{attribute 'GeneratedUsingTerminal: EL3314-0002-0016'}
{attribute addProperty BoxType "EL3314-0002-0016"}
{attribute addProperty Id "TC_Inputs_Channel_1AT %I*TC_Inputs_Channel_4521310411TC_Inputs_Channel_2AT %I*TC_Inputs_Channel_4521310411TC_Inputs_Channel_3AT %I*TC_Inputs_Channel_4521310411TC_Inputs_Channel_4AT %I*TC_Inputs_Channel_4521310411WcStateAT %I*WcState_9091E0EB2InfoDataAT %I*InfoData_94A18F5E2"}
{attribute addProperty CRC "1814089623"}
{attribute addProperty Size "48"}
TYPE EL3314_6C20CF97 EXTENDS EtcSlaveTerminalBase_947E5A46 :
STRUCT
	{attribute addProperty Name "TC_Inputs_Channel_1"}
	TC_Inputs_Channel_1 : TC_Inputs_Channel_45213104;
	{attribute addProperty Name "TC_Inputs_Channel_2"}
	TC_Inputs_Channel_2 : TC_Inputs_Channel_45213104;
	{attribute addProperty Name "TC_Inputs_Channel_3"}
	TC_Inputs_Channel_3 : TC_Inputs_Channel_45213104;
	{attribute addProperty Name "TC_Inputs_Channel_4"}
	TC_Inputs_Channel_4 : TC_Inputs_Channel_45213104;
	{attribute addProperty Name "WcState"}
	WcState : WcState_9091E0EB;
	{attribute addProperty Name "InfoData"}
	InfoData : InfoData_94A18F5E;
END_STRUCT
END_TYPE

(* stored: Version 1.2.0.0, ProductVersion 3.1.4024.9
   DUT EL3314_6C20CF97: Id {fd5a2d7d-3d27-4d71-bdda-629d7bba84dd} *)
